Yaskawa INFORM job: SKRZYNIA_4040_90_STOPNI_20BR.JBI

/JOB
//NAME SKRZYNIA_4040_90_STOPNI_20BR
///FOLDERNAME 02-SKRZYNIE_JOBS
//POS
///NPOS 315,315,0,24,0,0
///TOOL 0
///POSTYPE PULSE
///PULSE
C00000=0,-52280,40443,0,6876,0
C00001=82314,-24956,17040,59626,-27382,6248
C00002=93910,-8625,17040,59626,-43355,6248
C00003=98846,-1061,-42166,80308,-57081,-16120
C00004=100452,6057,-48127,85711,-56704,-21322
C00005=95573,33077,-33257,84645,-64023,-26851
C00006=94102,33899,-31937,85246,-63371,-26689
C00007=95573,33077,-33257,84645,-64023,-26851
C00008=94862,31071,-36438,85313,-63677,-27192
C00009=95573,33077,-33257,84645,-64023,-26851
C00010=95263,33142,-33256,84677,-63995,-26850
C00011=95263,33142,-33256,84677,-63995,-26850
C00012=94017,33843,-32133,85187,-63445,-26710
C00013=95263,33142,-33256,84677,-63995,-26850
C00014=94657,31439,-35966,85248,-63701,-27141
C00015=95263,33142,-33256,84677,-63995,-26850
C00016=95260,33144,-33256,84678,-63995,-26850
C00017=95260,33144,-33256,84678,-63995,-26850
C00018=94022,33838,-32141,85183,-63448,-26711
C00019=95260,33144,-33256,84678,-63995,-26850
C00020=94618,31343,-36117,85281,-63684,-27157
C00021=95260,33144,-33256,84678,-63995,-26850
C00022=95258,25631,32269,66559,-75499,-2416
C00023=95258,25631,32269,66559,-75499,-2416
C00024=94181,26497,33533,66410,-74896,-2191
C00025=95658,30184,39035,66708,-78559,-2356
C00026=95217,30377,39331,66881,-79841,-2558
C00027=95258,25631,32269,66559,-75499,-2416
C00028=98811,21047,-15512,99242,-81394,-20987
C00029=98811,21047,-15512,99242,-81394,-20987
C00030=97775,21639,-14693,99563,-80753,-20993
C00031=98811,21047,-15512,99242,-81394,-20987
C00032=98206,18840,-18520,99489,-81124,-21211
C00033=98811,21047,-15512,99242,-81394,-20987
C00034=97770,33535,58109,97477,-73223,-2907
C00035=97471,32489,56434,97533,-73096,-3098
C00036=96615,33295,57725,97337,-72490,-3014
C00037=97471,32489,56434,97533,-73096,-3098
C00038=97097,30483,53272,97662,-72975,-3435
C00039=97471,32489,56434,97533,-73096,-3098
C00040=98003,23984,26658,100907,-76471,-9645
C00041=97707,-10819,-23052,107304,-59718,-16318
C00042=94212,-35028,-34485,100444,-49148,-11285
C00043=48287,-44591,-17414,16172,-14532,25809
C00044=85348,-13130,13838,41209,-47455,8220
C00045=97395,20012,29210,69700,-74457,-9077
C00046=97055,28839,36684,71776,-79389,-10554
C00047=97055,28839,36684,71776,-79389,-10554
C00048=96058,29646,37897,71666,-78799,-10362
C00049=97055,28839,36684,71776,-79389,-10554
C00050=96570,26659,33451,71832,-78911,-10777
C00051=97055,28839,36684,71776,-79389,-10554
C00052=99260,22658,16753,92099,-78835,-1091
C00053=98782,22427,16945,92082,-78485,-960
C00054=98098,22870,17565,92116,-78014,-935
C00055=98782,22427,16945,92082,-78485,-960
C00056=98488,21195,15235,92147,-78307,-1085
C00057=98782,22427,16945,92082,-78485,-960
C00058=99953,7972,-32104,116782,-84999,-13620
C00059=94704,-17776,-58548,118507,-81680,-13914
C00060=60067,-64368,-72505,144806,-26050,-19168
C00061=60067,-50244,-32501,110603,-14199,-2207
C00062=63330,-26972,24478,18707,-56801,31483
C00063=95462,-31003,-33042,65414,-41305,6524
C00064=97787,-9790,-26685,81509,-54738,-4408
C00065=99864,21793,7359,80466,-76601,-6182
C00066=99753,21489,3165,89598,-79157,-3178
C00067=99071,20978,1948,89791,-78725,-3400
C00068=98206,21502,2669,89926,-78149,-3364
C00069=99071,20978,1948,89791,-78725,-3400
C00070=98727,19613,87,89895,-78511,-3524
C00071=99071,20978,1948,89791,-78725,-3400
C00072=99862,21793,7358,80466,-76600,-6182
C00073=98290,21024,6297,80683,-75539,-6194
C00074=97471,21541,7008,80756,-75007,-6115
C00075=98290,21024,6297,80683,-75539,-6194
C00076=97834,19245,3873,80814,-75197,-6333
C00077=98290,21024,6297,80683,-75539,-6194
C00078=98946,26804,31705,85784,-78857,-1423
C00079=98946,26804,31705,85784,-78857,-1423
C00080=98292,27270,32391,85749,-78414,-1361
C00081=98946,26804,31705,85784,-78857,-1423
C00082=98631,25349,29587,85839,-78632,-1590
C00083=98946,26804,31705,85784,-78857,-1423
C00084=94295,-1388,2615,87521,-55608,-1527
C00085=77022,-27457,-20499,75297,-20933,3764
///LIMIT ON
C00086=42754,-66126,12236,-1301,3231,7194
///LIMIT OFF
C00087=0,-52280,40443,0,6876,0
C00088=0,-52280,40443,0,6876,0
C00089=50509,-19000,10610,51503,-15997,-61182
C00090=50873,-17966,11417,52677,-16048,-61710
C00091=49459,-16590,12517,51258,-15158,-61190
C00092=50592,-16429,12648,53120,-15720,-61960
C00093=50873,-17966,11417,52677,-16048,-61710
C00094=50703,-18403,11066,52155,-16024,-61477
C00095=50703,-18403,11066,52155,-16024,-61477
C00096=49026,-16768,12358,50435,-14971,-60844
C00097=50653,-16371,12680,53228,-15754,-62008
C00098=50703,-18403,11066,52155,-16024,-61477
C00099=50704,-18401,11069,52157,-16021,-61478
C00100=50704,-20525,5414,58956,-14779,-64789
C00101=49025,-18889,6668,57745,-13658,-64384
C00102=50799,-18420,7036,60610,-14610,-65581
C00103=50704,-20525,5414,58956,-14779,-64789
C00104=51005,-17995,11387,52847,-16122,-61778
C00105=51005,-17995,11387,52847,-16122,-61778
C00106=49564,-16598,12501,51417,-15218,-61257
C00107=50954,-16306,12737,53719,-15902,-62212
C00108=51005,-17995,11387,52847,-16122,-61778
C00109=51030,-17981,11395,52891,-16138,-61796
C00110=51030,-17981,11395,52891,-16138,-61796
C00111=49401,-16396,12662,51265,-15114,-61201
C00112=50908,-16047,12947,53789,-15850,-62250
C00113=51030,-17981,11395,52891,-16138,-61796
C00114=50945,-18019,11363,52741,-16103,-61737
C00115=50945,-16980,14081,49884,-16761,-60338
C00116=49117,-15186,15539,47848,-15653,-59576
C00117=50939,-14679,15960,50992,-16487,-60881
C00118=50945,-18019,11363,52741,-16103,-61737
C00119=50945,-18019,11363,52741,-16103,-61737
C00120=50945,-18556,9943,54337,-15776,-62517
C00121=48967,-16606,11493,52445,-14510,-61829
C00122=51083,-15952,12027,56053,-15559,-63336
C00123=50945,-18556,9943,54337,-15776,-62517
C00124=50945,-18019,11363,52741,-16103,-61737
C00125=51350,-15183,18375,46705,-17991,-58719
C00126=49319,-13187,20053,44263,-16830,-57796
C00127=51236,-12618,20544,47529,-17647,-59142
C00128=51350,-15183,18375,46705,-17991,-58719
C00129=50028,-23690,-6096,22921,-31075,-54538
C00130=50670,-23735,-6923,24003,-30760,-55076
C00131=48518,-21492,-5254,21861,-29696,-54082
C00132=50138,-21068,-4928,23831,-30039,-55022
C00133=50670,-23735,-6923,24003,-30760,-55076
C00134=49763,-24225,-29961,22080,-30065,-59113
C00135=49763,-24225,-29961,22080,-30065,-59113
C00136=47727,-21550,-27874,20313,-29013,-58119
C00137=49271,-21042,-27466,22016,-29310,-59069
C00138=49763,-24225,-29961,22080,-30065,-59113
C00139=50713,-12366,-58367,41124,-17813,-74400
C00140=50713,-12366,-58367,41124,-17813,-74400
C00141=48934,-9522,-55687,39981,-16902,-73526
C00142=50242,-8975,-55157,41389,-17374,-74448
C00143=50713,-12366,-58367,41124,-17813,-74400
C00144=49763,-25421,-36239,24565,-26935,-60445
C00145=43547,-31626,-19626,5157,-49140,-52118
C00146=40154,-51179,-915,24203,-8234,-36524
C00147=0,-52280,40443,0,6876,0
C00148=0,-52280,40443,0,6876,0
C00149=0,-52280,40443,0,6876,0
C00150=82314,-24956,17040,59626,-27382,6248
C00151=93910,-8625,17040,59626,-43355,6248
C00152=98846,-1061,-42166,80308,-57081,-16120
C00153=100452,6057,-48127,85711,-56704,-21322
C00154=95564,34698,-34234,85516,-63941,-27819
C00155=93687,36612,-31081,84292,-64733,-27467
C00156=93711,36598,-31105,84282,-64744,-27471
C00157=95564,34698,-34234,85516,-63941,-27819
C00158=96930,32282,-32252,82595,-65816,-26305
C00159=93663,32611,-31732,84127,-64318,-26195
C00160=93663,32611,-31732,84127,-64318,-26195
C00161=96930,32282,-32252,82595,-65816,-26305
C00162=96528,-7533,-34932,76119,-53878,-10439
C00163=88377,-34186,-45291,67238,-52212,-2442
C00164=73560,-62084,7826,28695,-34737,3666
C00165=0,-52280,40443,0,6876,0
C00166=0,-36700,24612,-42871,-31823,-33862
C00167=44403,-30110,7154,24155,-23805,-45557
C00168=51347,-17798,16373,37641,-23556,-51399
C00169=51570,-17239,16856,38066,-23574,-51584
C00170=66126,-16365,3854,86555,-32059,-80935
C00171=60979,-15069,12509,70330,-26815,-71099
C00172=40431,-28773,9158,17648,-23273,-42875
C00173=0,-36700,24612,-42871,-31823,-33862
C00174=0,-52280,40443,0,6876,0
C00175=0,-52280,40443,0,6876,0
C00176=73560,-62084,7826,28695,-34737,3666
C00177=88377,-34186,-45291,67238,-52212,-2442
C00178=96920,-4461,-29697,76917,-56550,-10069
C00179=100432,21324,12575,83706,-77956,-7498
C00180=100432,21324,12575,83706,-77956,-7498
C00181=97224,21170,12361,83970,-75786,-7447
C00182=97224,21170,12361,83970,-75786,-7447
C00183=100432,21324,12575,83706,-77956,-7498
C00184=100432,21324,12575,83706,-77956,-7498
C00185=97481,25108,17890,83512,-78432,-7131
C00186=97624,25049,17805,83504,-78528,-7141
C00187=100432,21324,12575,83706,-77956,-7498
C00188=99336,18440,8642,84276,-74234,-7647
C00189=97735,24994,14595,85350,-78994,-5109
C00190=97744,25074,13580,86004,-79195,-4385
C00191=99336,18440,8642,84276,-74234,-7647
C00192=98746,26047,40390,96212,-73340,-2686
C00193=96511,23274,36200,96292,-71976,-3182
C00194=96511,27155,48340,94664,-71177,-571
C00195=99747,18296,13811,99163,-76345,-8478
C00196=99017,774,-48740,120026,-82763,-23886
C00197=82685,-42461,-85506,125714,-59125,-24709
///LIMIT ON
C00198=37721,-67612,11381,1325,-438,7850
///LIMIT OFF
C00199=37164,-60659,6466,13301,-5027,-19773
C00200=45362,-39990,2831,27538,-17767,-40935
C00201=57189,-26834,-7130,38780,-31731,-51561
C00202=63456,-14144,8594,45591,-40850,-50620
C00203=63236,-24074,-40908,65964,-30880,-63215
C00204=57189,-26834,-7130,38780,-31731,-51561
C00205=41180,-61187,4729,17280,-8498,-23442
C00206=0,-52280,40443,0,6876,0
C00207=0,-52280,40443,0,6876,0
///LIMIT ON
C00208=37721,-67612,11381,1325,-438,7850
///LIMIT OFF
C00209=43180,-50572,-20637,6552,-29302,38834
C00210=69362,-40002,-13521,39754,-33332,24421
C00211=86483,-21864,2840,55410,-40116,17549
C00212=99420,-11049,13736,67201,-51390,13904
C00213=92855,-5018,12828,77373,-48606,10660
C00214=98199,21452,7696,88481,-78015,-298
C00215=98177,26799,35147,85763,-78047,6724
C00216=100920,18905,27694,85174,-73370,7184
C00217=94483,-7610,-22783,94358,-54968,-958
C00218=98124,-17779,-18471,95902,-51295,3087
C00219=88943,-29687,-12397,76321,-42166,11919
C00220=82008,-39290,-17962,63915,-40768,19941
C00221=56258,-38103,3288,28818,-33580,-23051
C00222=41438,-37635,17580,13151,-29920,-38779
C00223=54964,-26842,8528,44141,-23181,-52038
C00224=50761,-21373,7883,46957,-18149,-54038
C00225=65101,-17441,-4948,103100,-32246,-89309
C00226=65181,-6263,27418,81207,-31059,-77222
C00227=56762,-20631,11812,69834,-24329,-69917
C00228=46096,-45842,-2681,20981,-19497,-36310
C00229=41180,-61187,4729,17280,-8498,-23442
C00230=0,-52280,40443,0,6876,0
C00231=0,-52280,40443,0,6876,0
///LIMIT ON
C00232=37721,-67612,11381,1325,-438,7850
///LIMIT OFF
C00233=43180,-50572,-20637,6552,-29302,38834
C00234=79425,-37128,-15462,51820,-35721,18807
C00235=92377,-29666,-26166,73570,-38078,7008
C00236=97441,-6012,-18634,86114,-58345,-2339
C00237=98864,-2001,-14672,90389,-62789,-3799
C00238=98767,21176,13691,87588,-77304,-2577
C00239=98123,23617,17097,87345,-78645,-2335
C00240=97979,23711,17231,87352,-78549,-2326
C00241=98864,-2001,-14672,90389,-62789,-3799
C00242=100472,-329,-13432,98539,-67097,-6304
C00243=92822,-26306,-37175,103295,-43881,-7703
C00244=68601,-52593,-52127,95725,-25602,-3235
C00245=80632,-38079,-20908,64053,-45216,12949
C00246=43180,-50572,-20637,6552,-29302,38834
///LIMIT ON
C00247=37721,-67612,11381,1325,-438,7850
///LIMIT OFF
C00248=0,-52280,40443,0,6876,0
///LIMIT ON
C00249=23708,-46776,23536,16027,-4787,-19738
///LIMIT OFF
C00250=50917,-40459,4132,34421,-18173,-42391
C00251=51059,-36587,4608,36647,-19418,-45358
C00252=50113,-22729,10834,36393,-23396,-50963
C00253=62046,-17757,4067,79440,-27252,-76630
C00254=63763,-15682,7486,80006,-29481,-77057
C00255=50113,-22729,10834,36393,-23396,-50963
C00256=43180,-50572,-20637,6552,-29302,38834
C00257=79425,-37128,-15462,51820,-35721,18807
C00258=92377,-33385,-41303,83059,-36844,1354
C00259=97441,-6012,-18634,86114,-58345,-2339
C00260=98442,-3149,-15680,86092,-59018,-2413
C00261=97114,-5888,-18685,94010,-59218,-3940
C00262=99563,18710,13338,88899,-76218,-2010
C00263=98011,23070,19863,88505,-78125,-1416
C00264=98011,24865,28095,87725,-78063,621
C00265=100205,15202,-8793,101167,-79304,-9541
C00266=100471,12680,2182,89317,-73847,-3746
C00267=93923,-8883,-21959,92925,-54783,-4609
C00268=92822,-26306,-37175,103295,-43881,-7703
C00269=68601,-52593,-52127,95725,-25602,-3235
C00270=29449,-70637,-48792,-22650,-13229,-23678
C00271=49121,-28282,-35458,21895,-29219,-59001
C00272=50484,-13386,-55713,36158,-19724,-71897
C00273=55938,-10187,-55661,55618,-22248,-82832
C00274=57381,15206,-57369,78100,-21009,-89969
C00275=50484,-13386,-55713,36158,-19724,-71897
C00276=49763,-25421,-36239,24565,-26935,-60445
C00277=50529,-22709,-3778,22940,-31995,-54502
C00278=45389,-28224,4312,35967,-15579,-54278
C00279=40154,-51179,-915,24203,-8234,-36524
C00280=0,-52280,40443,0,6876,0
C00281=0,-52280,40443,0,6876,0
///LIMIT ON
C00282=37721,-67612,11381,1325,-438,7850
///LIMIT OFF
C00283=43181,-50571,-20637,6551,-29300,38834
C00284=92325,-23846,-7228,63960,-40898,12897
C00285=85232,-2754,25377,50981,-49542,17626
C00286=95618,10017,30418,66150,-65403,10402
C00287=98328,26728,37723,75385,-78922,5377
C00288=99185,24817,27312,82025,-78466,1195
C00289=97766,23970,26102,82043,-77480,1145
C00290=97755,21890,16078,83086,-77017,-1370
C00291=100993,19573,16602,81480,-76704,-137
C00292=97883,29022,44703,72741,-79810,7156
C00293=99525,21729,17159,85870,-76787,-954
C00294=97991,25479,22462,85564,-79108,-597
C00295=97991,25479,22462,85564,-79108,-597
C00296=99525,21729,17159,85870,-76787,-954
C00297=99525,21703,17016,85886,-76785,-991
C00298=98063,26874,26717,84040,-79605,457
C00299=97834,25035,16764,84912,-79171,-2109
C00300=100039,22069,12584,85154,-78124,-2393
C00301=100072,10223,-2816,88932,-70713,-3891
C00302=99051,-8427,5223,77933,-54888,7183
C00303=82477,-27884,-1524,62699,-44420,15528
C00304=0,-52278,40443,0,6872,5
///LIMIT ON
C00305=23708,-46776,23536,16027,-4787,-19738
///LIMIT OFF
C00306=50917,-40459,4132,34421,-18173,-42391
C00307=49876,-21948,7530,68838,-10324,-59148
C00308=46721,-18942,9765,68167,-8197,-59205
C00309=59201,-15579,-1575,118679,-27419,-88015
C00310=59026,-13967,7015,105262,-23828,-78151
C00311=45927,-22803,4403,78462,-8511,-64553
C00312=62498,-35400,-2607,72048,-19281,-59202
C00313=31287,-69981,-10850,7253,-6843,-20996
C00314=0,-52280,40443,0,6876,0
BC00000=395344
BC00001=352964
BC00002=352964
BC00003=386755
BC00004=352964
BC00005=376061
BC00006=376061
BC00007=376061
BC00008=376061
BC00009=376061
BC00010=422255
BC00011=422255
BC00012=422255
BC00013=422255
BC00014=422255
BC00015=422255
BC00016=468422
BC00017=468422
BC00018=468422
BC00019=468422
BC00020=468422
BC00021=468422
BC00022=444238
BC00023=444238
BC00024=444238
BC00025=444238
BC00026=444238
BC00027=444238
BC00028=490292
BC00029=490292
BC00030=490292
BC00031=490292
BC00032=490292
BC00033=490292
BC00034=457501
BC00035=457501
BC00036=457501
BC00037=457501
BC00038=457501
BC00039=457501
BC00040=457501
BC00041=457501
BC00042=441126
BC00043=606955
BC00044=621951
BC00045=680325
BC00046=678232
BC00047=678232
BC00048=678232
BC00049=678232
BC00050=678232
BC00051=678232
BC00052=711282
BC00053=711282
BC00054=711282
BC00055=711282
BC00056=711282
BC00057=711282
BC00058=712827
BC00059=712827
BC00060=764717
BC00061=764717
BC00062=736982
BC00063=830816
BC00064=824770
BC00065=827573
BC00066=781421
BC00067=781421
BC00068=781421
BC00069=781421
BC00070=781421
BC00071=781421
BC00072=826243
BC00073=826243
BC00074=826243
BC00075=826243
BC00076=826243
BC00077=826243
BC00078=825637
BC00079=825637
BC00080=825637
BC00081=825637
BC00082=825637
BC00083=825637
BC00084=807693
BC00085=815028
BC00086=719510
BC00087=673544
BC00088=673544
BC00089=749807
BC00090=795890
BC00091=795890
BC00092=795890
BC00093=795890
BC00094=738548
BC00095=738548
BC00096=738548
BC00097=738548
BC00098=738548
BC00099=672663
BC00100=672663
BC00101=672663
BC00102=672663
BC00103=672663
BC00104=615008
BC00105=615008
BC00106=615008
BC00107=615008
BC00108=615008
BC00109=549905
BC00110=549905
BC00111=549905
BC00112=549905
BC00113=549905
BC00114=492580
BC00115=492580
BC00116=492580
BC00117=492580
BC00118=492580
BC00119=427066
BC00120=427066
BC00121=427066
BC00122=427066
BC00123=427066
BC00124=369647
BC00125=369647
BC00126=369647
BC00127=369647
BC00128=369647
BC00129=367378
BC00130=367378
BC00131=367378
BC00132=367378
BC00133=367378
BC00134=367378
BC00135=367378
BC00136=367378
BC00137=367378
BC00138=367378
BC00139=367378
BC00140=367378
BC00141=367378
BC00142=367378
BC00143=367378
BC00144=367378
BC00145=370159
BC00146=441050
BC00147=441050
BC00148=691458
BC00149=352964
BC00150=352964
BC00151=352964
BC00152=389827
BC00153=405188
BC00154=383772
BC00155=383772
BC00156=376148
BC00157=383772
BC00158=423163
BC00159=423163
BC00160=415475
BC00161=423163
BC00162=450041
BC00163=450041
BC00164=450041
BC00165=450041
BC00166=490644
BC00167=563016
BC00168=619936
BC00169=620614
BC00170=620150
BC00171=677247
BC00172=681587
BC00173=490644
BC00174=400994
BC00175=450041
BC00176=450041
BC00177=450041
BC00178=493267
BC00179=451598
BC00180=367111
BC00181=367111
BC00182=359499
BC00183=367111
BC00184=428582
BC00185=428582
BC00186=436302
BC00187=428582
BC00188=474694
BC00189=474702
BC00190=482470
BC00191=474694
BC00192=465890
BC00193=465890
BC00194=465890
BC00195=465890
BC00196=485423
BC00197=511514
BC00198=558282
BC00199=469376
BC00200=406602
BC00201=359905
BC00202=359905
BC00203=339797
BC00204=359905
BC00205=431999
BC00206=431999
BC00207=640937
BC00208=640937
BC00209=640937
BC00210=553973
BC00211=553967
BC00212=553967
BC00213=553967
BC00214=586920
BC00215=570679
BC00216=570679
BC00217=592240
BC00218=592240
BC00219=567686
BC00220=548194
BC00221=525052
BC00222=490703
BC00223=488588
BC00224=497390
BC00225=498168
BC00226=534717
BC00227=542091
BC00228=444406
BC00229=468922
BC00230=455634
BC00231=640937
BC00232=640937
BC00233=640937
BC00234=640937
BC00235=640937
BC00236=640937
BC00237=648365
BC00238=648365
BC00239=648365
BC00240=656045
BC00241=648365
BC00242=658303
BC00243=658303
BC00244=658303
BC00245=691207
BC00246=703131
BC00247=640937
BC00248=640937
BC00249=674716
BC00250=698935
BC00251=710701
BC00252=744351
BC00253=744351
BC00254=802868
BC00255=744351
BC00256=640937
BC00257=640937
BC00258=640937
BC00259=640937
BC00260=723517
BC00261=712075
BC00262=710772
BC00263=710772
BC00264=710772
BC00265=710772
BC00266=694536
BC00267=694444
BC00268=627581
BC00269=627581
BC00270=436090
BC00271=367378
BC00272=367378
BC00273=367378
BC00274=367381
BC00275=367378
BC00276=367378
BC00277=367378
BC00278=367374
BC00279=441050
BC00280=441050
BC00281=640937
BC00282=640937
BC00283=806788
BC00284=800422
BC00285=789823
BC00286=796863
BC00287=808786
BC00288=771476
BC00289=771476
BC00290=771476
BC00291=771185
BC00292=808786
BC00293=831813
BC00294=831813
BC00295=839479
BC00296=831813
BC00297=794344
BC00298=794344
BC00299=794344
BC00300=794344
BC00301=800112
BC00302=773022
BC00303=753838
BC00304=655351
BC00305=470174
BC00306=360196
BC00307=360196
BC00308=360196
BC00309=361315
BC00310=420934
BC00311=419944
BC00312=419842
BC00313=650116
BC00314=650116
///POSTYPE BASE
///RECTAN
///RCONF 1,0,0,0,0,0,0,0,0,0,0,0,0,0,0,0,0,0,0,0,0,0,0,0
P00006=0.000,0.000,0.000,0.0000,0.0000,0.0000
///RCONF 0,0,0,0,0,0,0,0,0,0,0,0,0,0,0,0,0,0,0,0,0,0,0,0
P00058=0.000,0.000,3.000,0.0000,0.0000,0.0000
///RCONF 1,0,0,0,0,0,0,0,0,0,0,0,0,0,0,0,0,0,0,0,0,0,0,0
P00300=-0.036,-1.505,2.318,0.0000,0.0000,0.0000
P00301=0.046,-2.112,7.779,0.0000,0.0000,0.0000
P00302=-0.180,-2.409,6.326,0.0000,0.0000,0.0000
///RCONF 0,0,0,0,0,0,0,0,0,0,0,0,0,0,0,0,0,0,0,0,0,0,0,0
P00303=-0.004,-1.437,-4.584,0.0000,0.0000,0.0000
P00304=0.028,-1.666,-4.234,0.0000,0.0000,0.0000
P00305=-0.003,-1.920,-3.501,0.0000,0.0000,0.0000
P00307=0.019,-2.151,-5.077,0.0000,0.0000,0.0000
P00308=-0.003,-2.092,-4.888,0.0000,0.0000,0.0000
P00309=-0.040,-2.205,-4.992,0.0000,0.0000,0.0000
P00310=-0.006,-2.490,-5.925,0.0000,0.0000,0.0000
P00311=-0.007,-2.079,-5.307,0.0000,0.0000,0.0000
P00351=13.563,-0.027,-0.653,0.0000,0.0000,0.0000
P00352=13.252,-0.027,-0.827,0.0000,0.0000,0.0000
P00353=10.971,-0.082,0.776,0.0000,0.0000,0.0000
P00354=-0.024,2.508,-1.824,0.0000,0.0000,0.0000
P00355=-0.001,2.528,-1.131,0.0000,0.0000,0.0000
P00356=-0.034,2.921,-0.262,0.0000,0.0000,0.0000
P00357=0.003,3.386,-0.091,0.0000,0.0000,0.0000
P00358=0.014,3.037,-0.020,0.0000,0.0000,0.0000
P00359=-0.005,2.731,0.912,0.0000,0.0000,0.0000
P00360=-0.011,3.412,0.438,0.0000,0.0000,0.0000
P00361=0.018,3.050,1.253,0.0000,0.0000,0.0000
//INST
///DATE 2025/03/28 12:19
///ATTR SC,RW
///GROUP1 RB1,BS1
NOP
CALL JOB:MOVE_INTO_TUNNEL
MOVJ C00000 BC00000 VJ=10.00
MOVJ C00001 BC00001 VJ=30.00
MOVJ C00002 BC00002 VJ=30.00
MOVL C00003 BC00003 V=500.0
COMM MOVJ C00004 BC00004 VJ=30.00
COMM '------------------------
COMM 'W65.3
COMM '------------------------
COMM MOVL C00005 BC00005 V=333.3 PL=0
COMM REFP 3 C00006 BC00006
COMM CALL JOB:SEARCH-R1
COMM SET P0300 P0006
COMM SFTON P0300
COMM MOVL C00007 BC00007 V=333.3 PL=0
COMM REFP 3 C00008 BC00008
COMM CALL JOB:SEARCH-R1
COMM SET P0300 P0006
COMM SFTON P0300
COMM MOVL C00009 BC00009 V=333.3 PL=0
COMM SFTOF
'------------------------
'W65.5
'------------------------
MOVL C00010 BC00010 V=500.0
MOVL C00011 BC00011 V=333.3 PL=0
REFP 3 C00012 BC00012
CALL JOB:SEARCH-R1
SET P0301 P0006
SFTON P0301
MOVL C00013 BC00013 V=333.3 PL=0
REFP 3 C00014 BC00014
CALL JOB:SEARCH-R1
SET P0301 P0006
SFTON P0301
MOVL C00015 BC00015 V=333.3 PL=0
SFTOF
'------------------------
'W65.7
'------------------------
MOVL C00016 BC00016 V=500.0
MOVL C00017 BC00017 V=333.3 PL=0
REFP 3 C00018 BC00018
CALL JOB:SEARCH-R1
SET P0302 P0006
SFTON P0302
MOVL C00019 BC00019 V=333.3 PL=0
REFP 3 C00020 BC00020
CALL JOB:SEARCH-R1
SET P0302 P0006
SFTON P0302
MOVL C00021 BC00021 V=500.0 PL=0
SFTOF
'------------------------
'W65.10
'------------------------
MOVL C00022 BC00022 V=500.0
MOVL C00023 BC00023 V=333.3 PL=0
REFP 3 C00024 BC00024
CALL JOB:SEARCH-R1
SET P0303 P0006
SFTON P0303
MOVL C00025 BC00025 V=333.3 PL=0
REFP 3 C00026 BC00026
CALL JOB:SEARCH-R1
SET P0303 P0006
SFTON P0303
MOVL C00027 BC00027 V=333.3 PL=0
SFTOF
'------------------------
'W65.12
'------------------------
MOVL C00028 BC00028 V=500.0
MOVL C00029 BC00029 V=333.3 PL=0
REFP 3 C00030 BC00030
CALL JOB:SEARCH-R1
SET P0304 P0006
SFTON P0304
MOVL C00031 BC00031 V=333.3 PL=0
REFP 3 C00032 BC00032
CALL JOB:SEARCH-R1
SET P0304 P0006
SFTON P0304
MOVL C00033 BC00033 V=333.3 PL=0
SFTOF
'------------------------
'W65.15
'------------------------
MOVL C00034 BC00034 V=500.0
MOVL C00035 BC00035 V=333.3 PL=0
REFP 3 C00036 BC00036
CALL JOB:SEARCH-R1
SET P0305 P0006
SFTON P0305
MOVL C00037 BC00037 V=333.3 PL=0
REFP 3 C00038 BC00038
CALL JOB:SEARCH-R1
SET P0305 P0006
SFTON P0305
MOVL C00039 BC00039 V=333.3 PL=0
SFTOF
'------------------------
'W65.17
'------------------------
MOVL C00040 BC00040 V=500.0
MOVL C00041 BC00041 V=333.3
MOVL C00042 BC00042 V=500.0
MOVJ C00043 BC00043 VJ=30.00
MOVL C00044 BC00044 V=500.0
MOVL C00045 BC00045 V=500.0
'------------------------
'W65.20
'------------------------
MOVL C00046 BC00046 V=500.0
MOVL C00047 BC00047 V=333.3 PL=0
REFP 3 C00048 BC00048
CALL JOB:SEARCH-R1
SET P0307 P0006
SFTON P0307
MOVL C00049 BC00049 V=333.3 PL=0
REFP 3 C00050 BC00050
CALL JOB:SEARCH-R1
SET P0307 P0006
SFTON P0307
MOVL C00051 BC00051 V=500.0 PL=0
SFTOF
'------------------------
'W65.23
'------------------------
MOVL C00052 BC00052 V=500.0
MOVL C00053 BC00053 V=333.3 PL=0
REFP 3 C00054 BC00054
CALL JOB:SEARCH-R1
SET P0308 P0006
SFTON P0308
MOVL C00055 BC00055 V=333.3 PL=0
REFP 3 C00056 BC00056
CALL JOB:SEARCH-R1
SET P0308 P0006
SFTON P0308
MOVL C00057 BC00057 V=500.0 PL=0
SFTOF
'------------------------
'W65.25
'------------------------
MOVL C00058 BC00058 V=333.3
MOVL C00059 BC00059 V=333.3
MOVL C00060 BC00060 V=500.0
MOVL C00061 BC00061 V=500.0
MOVL C00062 BC00062 V=250.0
MOVL C00063 BC00063 V=500.0
MOVL C00064 BC00064 V=500.0
MOVL C00065 BC00065 V=83.3
MOVL C00066 BC00066 V=500.0
MOVL C00067 BC00067 V=333.3 PL=0
REFP 3 C00068 BC00068
CALL JOB:SEARCH-R1
SET P0309 P0006
SFTON P0309
MOVL C00069 BC00069 V=333.3 PL=0
REFP 3 C00070 BC00070
CALL JOB:SEARCH-R1
SET P0309 P0006
SFTON P0309
MOVL C00071 BC00071 V=500.0 PL=0
SFTOF
'------------------------
'W65.28
'------------------------
MOVL C00072 BC00072 V=500.0
MOVL C00073 BC00073 V=333.3 PL=0
REFP 3 C00074 BC00074
CALL JOB:SEARCH-R1
SET P0310 P0006
SFTON P0310
MOVL C00075 BC00075 V=333.3 PL=0
REFP 3 C00076 BC00076
CALL JOB:SEARCH-R1
SET P0310 P0006
SFTON P0310
MOVL C00077 BC00077 V=333.3 PL=0
SFTOF
'------------------------
'W65.30
'------------------------
MOVL C00078 BC00078 V=500.0
MOVL C00079 BC00079 V=333.3 PL=0
REFP 3 C00080 BC00080
CALL JOB:SEARCH-R1
SET P0311 P0006
SFTON P0311
MOVL C00081 BC00081 V=333.3 PL=0
REFP 3 C00082 BC00082
CALL JOB:SEARCH-R1
SET P0311 P0006
SFTON P0311
MOVL C00083 BC00083 V=333.3 PL=0
SFTOF
MOVL C00084 BC00084 V=500.0
MOVL C00085 BC00085 V=500.0
MOVJ C00086 BC00086 VJ=30.00
MOVJ C00087 BC00087 VJ=30.00
MOVJ C00088 BC00088 VJ=30.00
'------------------------
MOVJ C00089 BC00089 VJ=30.00
MOVL C00090 BC00090 V=333.3 PL=0
REFP 3 C00091 BC00091
CALL JOB:SEARCH-R1
IMOV P0058 V=16.7
SET P0351 P0006
SFTON P0351
REFP 3 C00092 BC00092
CALL JOB:SEARCH-R1
SET P0351 P0006
SFTON P0351
MOVL C00093 BC00093 V=500.0 PL=0
SFTOF
'------------------------
'W254A L
'------------------------
MOVJ C00094 BC00094 VJ=30.00
MOVL C00095 BC00095 V=333.3 PL=0
REFP 3 C00096 BC00096
CALL JOB:SEARCH-R1
IMOV P0058 V=16.7
SET P0352 P0006
SFTON P0352
REFP 3 C00097 BC00097
CALL JOB:SEARCH-R1
SET P0352 P0006
SFTON P0352
MOVL C00098 BC00098 V=500.0 PL=0
SFTOF
'------------------------
'W250A P
'------------------------
MOVJ C00099 BC00099 VJ=30.00
MOVL C00100 BC00100 V=333.3 PL=0
REFP 3 C00101 BC00101
CALL JOB:SEARCH-R1
IMOV P0058 V=16.7
SET P0353 P0006
SFTON P0353
REFP 3 C00102 BC00102
CALL JOB:SEARCH-R1
SET P0353 P0006
SFTON P0353
MOVL C00103 BC00103 V=500.0 PL=0
SFTOF
'------------------------
'W250A L
'------------------------
MOVJ C00104 BC00104 VJ=30.00
MOVL C00105 BC00105 V=333.3 PL=0
REFP 3 C00106 BC00106
CALL JOB:SEARCH-R1
IMOV P0058 V=16.7
SET P0354 P0006
SFTON P0354
REFP 3 C00107 BC00107
CALL JOB:SEARCH-R1
SET P0354 P0006
SFTON P0354
MOVL C00108 BC00108 V=500.0 PL=0
SFTOF
'------------------------
'W253A P
'------------------------
MOVJ C00109 BC00109 VJ=30.00
MOVL C00110 BC00110 V=333.3 PL=0
REFP 3 C00111 BC00111
CALL JOB:SEARCH-R1
IMOV P0058 V=16.7
SET P0355 P0006
SFTON P0355
REFP 3 C00112 BC00112
CALL JOB:SEARCH-R1
SET P0355 P0006
SFTON P0355
MOVL C00113 BC00113 V=333.3 PL=0
SFTOF
'------------------------
'W253A L
'------------------------
MOVJ C00114 BC00114 VJ=30.00
MOVL C00115 BC00115 V=333.3 PL=0
REFP 3 C00116 BC00116
CALL JOB:SEARCH-R1
IMOV P0058 V=16.7
SET P0356 P0006
SFTON P0356
REFP 3 C00117 BC00117
CALL JOB:SEARCH-R1
SET P0356 P0006
SFTON P0356
MOVL C00118 BC00118 V=500.0 PL=0
SFTOF
'------------------------
'W256A P
'------------------------
MOVJ C00119 BC00119 VJ=30.00
MOVL C00120 BC00120 V=333.3 PL=0
REFP 3 C00121 BC00121
CALL JOB:SEARCH-R1
IMOV P0058 V=16.7
SET P0357 P0006
SFTON P0357
REFP 3 C00122 BC00122
CALL JOB:SEARCH-R1
SET P0357 P0006
SFTON P0357
MOVL C00123 BC00123 V=500.0 PL=0
SFTOF
'------------------------
'W256A L
'------------------------
MOVJ C00124 BC00124 VJ=30.00
MOVL C00125 BC00125 V=333.3 PL=0
REFP 3 C00126 BC00126
CALL JOB:SEARCH-R1
IMOV P0058 V=16.7
SET P0358 P0006
SFTON P0358
REFP 3 C00127 BC00127
CALL JOB:SEARCH-R1
SET P0358 P0006
SFTON P0358
MOVL C00128 BC00128 V=500.0 PL=0
SFTOF
'------------------------
'W252A P
'------------------------
MOVL C00129 BC00129 V=500.0
MOVL C00130 BC00130 V=333.3 PL=0
REFP 3 C00131 BC00131
CALL JOB:SEARCH-R1
IMOV P0058 V=16.7
SET P0359 P0006
SFTON P0359
REFP 3 C00132 BC00132
CALL JOB:SEARCH-R1
SET P0359 P0006
SFTON P0359
MOVL C00133 BC00133 V=333.3 PL=0
SFTOF
'------------------------
'W252A L
'------------------------
MOVL C00134 BC00134 V=500.0
MOVL C00135 BC00135 V=333.3 PL=0
REFP 3 C00136 BC00136
CALL JOB:SEARCH-R1
IMOV P0058 V=16.7
SET P0360 P0006
SFTON P0360
REFP 3 C00137 BC00137
CALL JOB:SEARCH-R1
SET P0360 P0006
SFTON P0360
MOVL C00138 BC00138 V=500.0 PL=0
SFTOF
COMM '------------------------
COMM 'W255A
COMM '------------------------
COMM MOVL C00139 BC00139 V=500.0
COMM MOVL C00140 BC00140 V=333.3 PL=0
COMM REFP 3 C00141 BC00141
COMM CALL JOB:SEARCH-R1
COMM IMOV P0058 V=16.7
COMM SET P0361 P0006
COMM SFTON P0361
COMM REFP 3 C00142 BC00142
COMM CALL JOB:SEARCH-R1
COMM SET P0361 P0006
COMM SFTON P0361
COMM MOVL C00143 BC00143 V=500.0 PL=0
COMM SFTOF
COMM MOVL C00144 BC00144 V=500.0
MOVJ C00145 BC00145 VJ=50.00
MOVJ C00146 BC00146 VJ=50.00
MOVJ C00147 BC00147 VJ=50.00
MOVJ C00148 BC00148 VJ=50.00
CALL JOB:FRONT_SEARCH_90ST-2_4040
MOVJ C00149 BC00149 VJ=50.00
MOVJ C00150 BC00150 VJ=40.00
MOVJ C00151 BC00151 VJ=30.00
MOVL C00152 BC00152 V=666.7
MOVJ C00153 BC00153 VJ=40.00
COMM '------------------------
COMM 'W65.3
COMM '------------------------
COMM SFTON P0300
COMM MOVL C00154 BC00154 V=500.0
COMM MOVL C00155 BC00155 V=333.3 PL=0
COMM MACRO1 MJ#(0) ARGF10
COMM ARCON
COMM MOVL C00156 BC00156 V=10.8
COMM ARCOF
COMM MOVL C00157 BC00157 V=166.7
COMM SFTOF
COMM '------------------------
COMM 'W65.5
COMM '------------------------
SFTON P0301
MOVL C00158 BC00158 V=333.3
MOVL C00159 BC00159 V=133.3 PL=0
MACRO1 MJ#(0) ARGF10
ARCON
MOVL C00160 BC00160 V=10.8
ARCOF
MOVL C00161 BC00161 V=166.7
SFTOF
MOVL C00162 BC00162 V=500.0
MOVL C00163 BC00163 V=333.3
MOVJ C00164 BC00164 VJ=25.00
MOVJ C00165 BC00165 VJ=50.00
'::::::::::::::::::::::::::::::::
'::::::::::::::::::::::::::::::::
'::::::::::::::::::::::::::::::::
'::::::::::::::::::::::::::::::::
'::::::::::::::::::::::::::::::::
MOVJ C00166 BC00166 VJ=50.00
MOVJ C00167 BC00167 VJ=50.00
MOVJ C00168 BC00168 VJ=50.00
'------------------------
'W250A
'------------------------
SFTON P0354
MOVL C00169 BC00169 V=333.3
MOVL C00170 BC00170 V=133.3 PL=0
MACRO1 MJ#(0) ARGF29
ARCON
SFTOF
SFTON P0353
MOVL C00171 BC00171 V=12.5
ARCOF
MOVL C00172 BC00172 V=166.7
SFTOF
MOVJ C00173 BC00173 VJ=50.00
MOVJ C00174 BC00174 VJ=50.00
MOVJ C00175 BC00175 VJ=50.00
MOVJ C00176 BC00176 VJ=50.00
MOVJ C00177 BC00177 VJ=50.00
MOVJ C00178 BC00178 VJ=20.00
MOVJ C00179 BC00179 VJ=10.00
'------------------------
'W65.7
'------------------------
SFTON P0302
'MOTOSIM PULSE LIMIT
MOVL C00180 BC00180 V=500.0
MOVL C00181 BC00181 V=133.3 PL=0
MACRO1 MJ#(0) ARGF30
ARCON
MOVL C00182 BC00182 V=11.7
ARCOF
MOVL C00183 BC00183 V=250.0
SFTOF
'------------------------
'W65.10
'------------------------
SFTON P0303
MOVL C00184 BC00184 V=500.0
MOVL C00185 BC00185 V=166.7 PL=0
ARCON
MOVL C00186 BC00186 V=11.7
ARCOF
MOVL C00187 BC00187 V=166.7
SFTOF
'------------------------
'W65.12
'------------------------
SFTON P0304
MOVL C00188 BC00188 V=333.3
MOVL C00189 BC00189 V=133.3 PL=0
MACRO1 MJ#(0) ARGF30
ARCON
MOVL C00190 BC00190 V=11.7
ARCOF
MOVL C00191 BC00191 V=166.7
SFTOF
'------------------------
'W65.15
'------------------------
SFTON P0305
MOVL C00192 BC00192 V=333.3
MOVL C00193 BC00193 V=166.7 PL=0
ARCON
MOVL C00194 BC00194 V=11.7
ARCOF
MOVL C00195 BC00195 V=166.7
SFTOF
MOVL C00196 BC00196 V=333.3
MOVL C00197 BC00197 V=500.0
MOVJ C00198 BC00198 VJ=50.00
MOVJ C00199 BC00199 VJ=50.00
MOVJ C00200 BC00200 VJ=50.00
'------------------------
'W252A
'------------------------
SFTON P0359
MOVL C00201 BC00201 V=500.0
MOVL C00202 BC00202 V=166.7 PL=0
MACRO1 MJ#(0) ARGF29
ARCON
SFTOF
SFTON P0358
MOVL C00203 BC00203 V=12.5
ARCOF
MOVL C00204 BC00204 V=250.0
SFTOF
MOVJ C00205 BC00205 VJ=50.00
MOVJ C00206 BC00206 VJ=80.00
MOVJ C00207 BC00207 VJ=80.00
MOVJ C00208 BC00208 VJ=50.00
MOVJ C00209 BC00209 VJ=50.00
MOVJ C00210 BC00210 VJ=25.00
MOVL C00211 BC00211 V=333.3
MOVL C00212 BC00212 V=333.3
'------------------------
'W65.17
'------------------------
MOVL C00213 BC00213 V=166.7
SFTON P0305
MOVL C00214 BC00214 V=166.7 PL=0
MACRO1 MJ#(0) ARGF30
ARCON
MOVL C00215 BC00215 V=11.7
ARCOF
SFTOF
MOVL C00216 BC00216 V=166.7
SFTOF
MOVL C00217 BC00217 V=250.0
MOVL C00218 BC00218 V=250.0
MOVL C00219 BC00219 V=333.3
MOVJ C00220 BC00220 VJ=25.00
'::::::::::::::::::::::::
'::::::::::::::::::::::::
'::::::::::::::::::::::::
'::::::::::::::::::::::::
'::::::::::::::::::::::::
'::::::::::::::::::::::::
'::::::::::::::::::::::::
'::::::::::::::::::::::::::::::::
'::::::::::::::::::::::::::::::::
'------------------------
'W61.17
'------------------------
'::::::::::::::::::::::::::::::::
'::::::::::::::::::::::::::::::::
'------------------------
'W253A
'------------------------
MOVJ C00221 BC00221 VJ=50.00
MOVJ C00222 BC00222 VJ=50.00
SFTON P0356
MOVL C00223 BC00223 V=333.3
MOVL C00224 BC00224 V=333.3
MOVL C00225 BC00225 V=166.7 PL=0
MACRO1 MJ#(0) ARGF29
ARCON
SFTOF
SFTON P0355
MOVL C00226 BC00226 V=12.5
ARCOF
MOVL C00227 BC00227 V=250.0
SFTOF
MOVJ C00228 BC00228 VJ=50.00
MOVJ C00229 BC00229 VJ=50.00
MOVJ C00230 BC00230 VJ=80.00
MOVJ C00231 BC00231 VJ=80.00
MOVJ C00232 BC00232 VJ=50.00
MOVJ C00233 BC00233 VJ=50.00
MOVJ C00234 BC00234 VJ=50.00
MOVJ C00235 BC00235 VJ=30.00
MOVJ C00236 BC00236 VJ=30.00
'------------------------
'W65.20
'------------------------
SFTON P0307
MOVL C00237 BC00237 V=333.3
MOVL C00238 BC00238 V=166.7
MOVL C00239 BC00239 V=166.7 PL=0
MACRO1 MJ#(0) ARGF30
ARCON
MOVL C00240 BC00240 V=11.7
ARCOF
MOVL C00241 BC00241 V=250.0
SFTOF
MOVL C00242 BC00242 V=333.3
MOVL C00243 BC00243 V=333.3
MOVL C00244 BC00244 V=333.3
MOVJ C00245 BC00245 VJ=50.00
MOVJ C00246 BC00246 VJ=50.00
MOVJ C00247 BC00247 VJ=50.00
MOVJ C00248 BC00248 VJ=50.00
MOVJ C00249 BC00249 VJ=50.00
MOVJ C00250 BC00250 VJ=50.00
SFTON P0352
MOVL C00251 BC00251 V=500.0
MOVL C00252 BC00252 V=500.0
MOVL C00253 BC00253 V=166.7 PL=0
MACRO1 MJ#(0) ARGF29
ARCON
SFTOF
SFTON P0351
MOVL C00254 BC00254 V=12.5
ARCOF
MOVL C00255 BC00255 V=333.3
SFTOF
MOVJ C00256 BC00256 VJ=50.00
MOVJ C00257 BC00257 VJ=50.00
MOVJ C00258 BC00258 VJ=50.00
MOVJ C00259 BC00259 VJ=30.00
MOVL C00260 BC00260 V=500.0
'------------------------
'W65.23
'------------------------
SFTON P0308
MOVL C00261 BC00261 V=333.3
MOVL C00262 BC00262 V=166.7
MOVL C00263 BC00263 V=133.3 PL=0
MACRO1 MJ#(0) ARGF30
ARCON
MOVL C00264 BC00264 V=11.7
ARCOF
MOVL C00265 BC00265 V=166.7
SFTOF
'------------------------
'W65.25
'------------------------
MOVL C00266 BC00266 V=500.0
MOVL C00267 BC00267 V=333.3
MOVL C00268 BC00268 V=500.0
MOVL C00269 BC00269 V=333.3
MOVJ C00270 BC00270 VJ=80.00
COMM '------------------------
COMM 'W255A
COMM MOVL C00271 BC00271 V=500.0
COMM MOVL C00272 BC00272 V=333.3
COMM SFTON P0361
COMM MOVL C00273 BC00273 V=133.3 PL=0
COMM MACRO1 MJ#(0) ARGF29
COMM ARCON
COMM MOVL C00274 BC00274 V=12.5
COMM ARCOF
COMM MOVL C00275 BC00275 V=250.0
COMM SFTOF
COMM MOVL C00276 BC00276 V=333.3
COMM MOVL C00277 BC00277 V=333.3
COMM MOVL C00278 BC00278 V=500.0
MOVJ C00279 BC00279 VJ=50.00
MOVJ C00280 BC00280 VJ=50.00
MOVJ C00281 BC00281 VJ=80.00
MOVJ C00282 BC00282 VJ=50.00
MOVJ C00283 BC00283 VJ=50.00
MOVL C00284 BC00284 V=333.3
'------------------------
'W31.28
'------------------------
SFTON P0310
MOVL C00285 BC00285 V=333.3
MOVL C00286 BC00286 V=333.3
MOVL C00287 BC00287 V=166.7
SFTON P0309
MOVL C00288 BC00288 V=500.0
MOVL C00289 BC00289 V=133.3 PL=0
ARCON
MOVL C00290 BC00290 V=11.7
ARCOF
MOVL C00291 BC00291 V=166.7
SFTOF
MOVL C00292 BC00292 V=250.0
SFTOF
'------------------------
'W31.30
'------------------------
SFTON P0311
MOVL C00293 BC00293 V=333.3
MOVL C00294 BC00294 V=133.3 PL=0
MACRO1 MJ#(0) ARGF30
ARCON
MOVL C00295 BC00295 V=11.7
ARCOF
MOVL C00296 BC00296 V=166.7
MOVL C00297 BC00297 V=333.3
SFTON P0310
MOVL C00298 BC00298 V=166.7
ARCON
MOVL C00299 BC00299 V=11.7
ARCOF
SFTOF
MOVL C00300 BC00300 V=166.7
MOVL C00301 BC00301 V=333.3
SFTOF
MOVL C00302 BC00302 V=500.0
MOVL C00303 BC00303 V=333.3
'::::::::::::::::::::::::
'::::::::::::::::::::::::
'::::::::::::::::::::::::
'::::::::::::::::::::::::
'::::::::::::::::::::::::
'::::::::::::::::::::::::
'::::::::::::::::::::::::
MOVJ C00304 BC00304 VJ=50.00 PL=0
MOVJ C00305 BC00305 VJ=80.00
MOVJ C00306 BC00306 VJ=80.00
SFTON P0358
MOVL C00307 BC00307 V=333.3
MOVL C00308 BC00308 V=250.0
MOVL C00309 BC00309 V=166.7 PL=0
MACRO1 MJ#(0) ARGF29
ARCON
SFTOF
SFTON P0357
MOVL C00310 BC00310 V=12.5
ARCOF
MOVL C00311 BC00311 V=333.3
SFTOF
MOVJ C00312 BC00312 VJ=50.00
MOVJ C00313 BC00313 VJ=50.00
MOVJ C00314 BC00314 VJ=80.00
CALL JOB:FRONT_WELD_90ST-2_4040
CALL JOB:MOVE_OUT_OF_TUNNEL
END
